// AnalogInReal FB to read and scale a single REAL input
// Set bit 3 (Options.3) to true to enable scaling based on +/-7812500 instead of legacy range values +/-838860x
// NoOfDigits per default set to 3... 
FUNCTION_BLOCK AnalogInREAL EXTENDS EcSlaveInfoDataExt
VAR_INPUT
	Offset													:	LREAL 		:= 0.0;
	MinValue												: 	LREAL 		:= 0.0;
	MaxValue												: 	LREAL 		:= 0.0;
	NoOfDigits												: 	INT(0..10)	:= 0; //number of decimal digits of scaled Q variable 
	OutOnError												:	LREAL 		:= 0.000000000000000001;
{attribute 'displaymode':='binary'}     	            	
	Options													:	BYTE  		:= 2#0000_0000;
END_VAR                 									
VAR                        
END_VAR                                 	            	
VAR_OUTPUT                              	            	                                       	
	Q														:	LREAL;//scaled result value
	In											AT  %I* 	: 	REAL; //Hardware Input
	{attribute 'displaymode':='binary'}     	            	
	Status										AT  %I*		:	WORD := 2#00000000_00000000;	//Terminal status (2 bytes)
END_VAR

(* Read single REAL value from terminal and scale to user units				*)
(****************************************************************************)

(* Scaling ******************************************************************)
	IF MaxValue <> MinValue 
	THEN			
		IF NOT Options.3
		THEN
			Q 	 											:= Offset + Scale(TO_LREAL(In), -8388608.0, 8388607.0, MinValue , MaxValue);
		ELSE
			Q 	 											:= Offset + Scale(TO_LREAL(In),  -7812500.0, 7812500.0, MinValue , MaxValue);		
		END_IF	
		
		IF NoOfDigits > 0
		THEN
			Q												:= TO_FMLREAL(Q,NoOfDigits);
		END_IF
	
	ELSIF NoOfDigits > 0 (* Bsp PT100 *)
	THEN
		Q													:= Offset + TO_FMLREAL(In,NoOfDigits);
		
	ELSE  													
		Q 													:= 0.0;
	END_IF

(****************************************************************************)

{attribute 'monitoring' := 'call'}
PROPERTY PUBLIC Error : BOOL
GET
Error					:= Status.6 OR MinValue = MaxValue AND NoOfDigits = 0;
END_GET
END_PROPERTY

{attribute 'monitoring' := 'call'}
PROPERTY PUBLIC Limit_1 : BYTE
GET
Limit_1.0					:= Status.2;
Limit_1.1					:= Status.3;
END_GET
END_PROPERTY

{attribute 'monitoring' := 'call'}
PROPERTY PUBLIC Limit_2 : BYTE
GET
Limit_2.0					:= Status.4;
Limit_2.1					:= Status.5;
END_GET
END_PROPERTY

PROPERTY PUBLIC optEnableScaleExtRangeMode : bool
GET
optEnableScaleExtRangeMode := Options.3;
END_GET
SET
Options.3 := optEnableScaleExtRangeMode;
END_SET
END_PROPERTY

{attribute 'monitoring' := 'call'}
PROPERTY PUBLIC Overrange : BOOL
GET
Overrange 			:= Status.1;
END_GET
END_PROPERTY

{attribute 'monitoring' := 'call'}
PROPERTY PUBLIC TareActive : BOOL
GET
TareActive					:= Status.11;
END_GET
END_PROPERTY

{attribute 'monitoring' := 'call'}
PROPERTY PUBLIC TxPDOState : BOOL
GET
TxPDOState					:= Status.14; //True if not valid
END_GET
END_PROPERTY

{attribute 'monitoring' := 'call'}
PROPERTY PUBLIC TxPDOToggle : BOOL
GET
TxPDOToggle							:= Status.15;
END_GET
END_PROPERTY

{attribute 'monitoring' := 'call'}
PROPERTY PUBLIC Underrange : BOOL
GET
Underrange 			:= Status.0;
END_GET
END_PROPERTY

END_FUNCTION_BLOCK

(* stored: Version 1.1.0.1, ProductVersion 3.1.4024.13
   POU AnalogInREAL: Id {3c8146b7-b009-4d8e-b324-0bfa5d735887}, SpecialFunc None
   Property Error: Id {ca453eed-6a9f-4737-960b-d2f3d15a46de}
   Get Get: Id {2ba81606-cdb6-44cc-b1a5-04dc9879ca77}
   Property Limit_1: Id {501e4239-6301-4fc9-8bef-9bf3dfafa22c}
   Get Get: Id {847b48ef-7ae0-46be-a39a-5101853c5ec3}
   Property Limit_2: Id {6224c693-1743-4d90-92f9-92dd613e5c4b}
   Get Get: Id {fca64313-61cf-4140-9263-f24d9d11df48}
   Property optEnableScaleExtRangeMode: Id {c7d501b6-cf7a-4a92-a5b5-9de8a39da864}
   Get Get: Id {79270da5-3e35-4d20-83ee-eb362bed1779}
   Set Set: Id {ba1ed693-72fb-489a-86b4-df7ffd35f0fe}
   Property Overrange: Id {61228141-9164-4268-a087-01a4d0b69bd2}
   Get Get: Id {4314db14-2e15-4d9b-8bac-e543be1e4d74}
   Property TareActive: Id {8eb79860-5ee9-45b4-92dd-50fbaffe8b5d}
   Get Get: Id {4e00d335-8bd8-4e2b-8d42-d1219f9c9a57}
   Property TxPDOState: Id {421ee044-bb0d-40be-8fa5-14cca3f8664a}
   Get Get: Id {28fb0f06-1441-43b4-876b-5a6134a8d2e5}
   Property TxPDOToggle: Id {bce3c13d-5bf4-4b53-82e4-56e171f5645e}
   Get Get: Id {029cd1fa-10ea-4e61-847c-e831bc596d48}
   Property Underrange: Id {4c21e517-afa9-4645-b002-c95d7ea9356a}
   Get Get: Id {859565e4-2188-4706-9d53-d7975233fd3f} *)
